PROGRAM MAIN
VAR
	// Transports — call before the devices that use them
	fbTcp          : FB_MbTransportTcp;
	fbRs485        : FB_MbTransportRtu;

	// Devices
	fbDemo         : FB_Mb_DiagDemo;
	fbMeter        : FB_Mb_TestGood;
	fbTemp		   : FB_ModbusDevice;

	// Write handshake example
	fSetpointCmd   : LREAL;
	bWriteSetpoint : BOOL;
END_VAR

// ---- Transports ----
fbTcp(sHost := GVL_Site.sTcpHost, nPort := GVL_Site.nTcpPort);
fbRs485(pComIn := ADR(GVL_IO.stEl6In1), pComOut := ADR(GVL_IO.stEl6Out1), nSizeComIn := SIZEOF(GVL_IO.stEl6In1));

// ---- Devices ----
fbDemo(itfTransport := fbTcp,   nUnitId := GVL_Site.nDemoUnit,  bEnable := TRUE);
fbMeter(itfTransport := fbRs485, nUnitId := GVL_Site.nMeterUnit, bEnable := TRUE, sLogName := 'FlowMeter_Inlet');

// ---- Write handshake: set fSetpointCmd, pulse bWriteSetpoint ----
IF bWriteSetpoint AND NOT fbDemo.Setpoint.bWriteReq AND NOT fbDemo.Setpoint.bWriteBusy THEN
	fbDemo.Setpoint.fWriteValue := fSetpointCmd;
	fbDemo.Setpoint.bWriteReq   := TRUE;
END_IF

IF fbDemo.Setpoint.bWriteDone OR fbDemo.Setpoint.bWriteErr THEN
	fbDemo.Setpoint.bWriteReq := FALSE;
	bWriteSetpoint            := FALSE;
END_IF

END_PROGRAM

(* stored: Version 1.1.0.1
   POU MAIN: Id {d2604a9c-1e7f-4fbb-88a2-792b3944e14d}, SpecialFunc None *)
